Omron CX-Programmer project NewProject (CX-Programmer 9.73)

# PLC Omron_test: CJ2M CPU11

## Global symbols (name address type ; comment)
0.00 BOOL  ; BTN
100.00 BOOL  ; RED
100.01 BOOL  ; YELLOW

## Program NewProgram1 (cyclic task 0)

### Section Section1

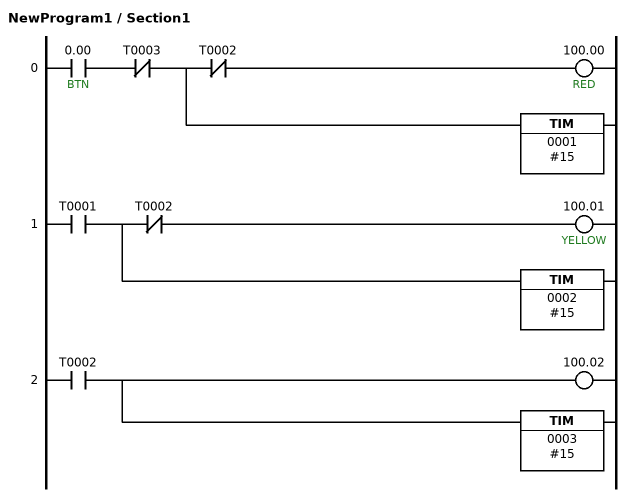
; rung 0
LD 0.00  ; BTN
ANDNOT T0003
OUT TR0
ANDNOT T0002
OUT 100.00  ; RED
LD TR0
TIM 0001 #15
; rung 1
LD T0001
OUT TR0
ANDNOT T0002
OUT 100.01  ; YELLOW
LD TR0
TIM 0002 #15
; rung 2
LD T0002
OUT 100.02
TIM 0003 #15

### Section END
; rung 0
END(001)